// TIA Portal V17 export
// export: Created 2024-08-26T21:10:49.0093194Z, ExportSetting WithDefaults, DisplayName Totally Integrated Automation Portal, DisplayVersion V17 Update 7, DisplayName TIA Portal Openness, DisplayVersion V17 Update 7, DisplayName TIA Portal Version Control Interface, DisplayVersion V17, DisplayName SINAMICS Startdrive Advanced, DisplayVersion V17 SP2, DisplayName SINAMICS Startdrive G110M, G120, G120C, G120D, G120P, G115D, DisplayVersion V17 SP2, DisplayName SINAMICS Startdrive G130, G150, S120, S150, SINAMICS MV, S210, DisplayVersion V17 SP2, DisplayName STEP 7 Professional, DisplayVersion V17 Update 7, DisplayName STEP 7 Safety, DisplayVersion V17 Update 6, DisplayName WinCC Advanced / Unified PC, DisplayVersion V17 Update 7
FUNCTION "smartLightControl" : Void   // FC7, LAD
{ S7_Optimized_Access := 'TRUE' }
VERSION : 0.1
// stored: AutoNumber true, IsIECCheckEnabled false, SetENOAutomatically false, UDAEnableTagReadback false
   VAR_INPUT
      iRedSolid : Bool;
      iRedBlinking : Bool;
      iAmbarSolid : Bool;
      iAmbarBlinking : Bool;
      iGreenSolid : Bool;
      iGreenBlinking : Bool;
      iBlueSolid : Bool;
      iBlueBlinking : Bool;
   END_VAR
   VAR_OUTPUT
      byte0ColorAndBlink : Byte;   // Segment 1 and 2
      byte1ColorAndBlink : Byte;   // Segment 3
      byte2BuzzerType : Byte;
      byte3ModeSelect : Byte;
      byte4NumberOfSegments : Byte;
      byte5BlinkMode : Byte;
      byte6BlinkFreq : Byte;
      byte7BuzzerVolume : Byte;
   END_VAR
   VAR_TEMP
      segment1Color : Byte;
      segment2Color : Byte;
      segment3Color : Byte;
      colorsToDisplay : Word;
      numberOfColorsToDisplay : UInt;
      colorToAddToQueue : Word;
      positionsToMove : UInt;
   END_VAR
   VAR CONSTANT
      redColor : Byte := 2#0010;
      blueColor : Byte := 2#0100;
      ambarColor : Byte := 2#0101;
      greenColor : Byte := 2#0001;
      redBlinkingColor : Byte := 2#1010;
      blueBlinkingColor : Byte := 2#1100;
      ambarBlinkingColor : Byte := 2#1101;
      greenBlinkingColor : Byte := 2#1001;
   END_VAR
BEGIN

REGION Network 1: INIT
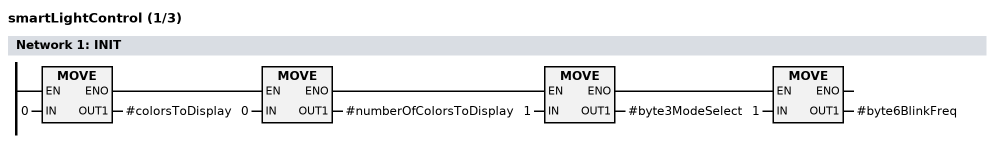
   RUNG wire#powerrail
      Move(in := 0, out1 => #colorsToDisplay)
      Move(in := 0, out1 => #numberOfColorsToDisplay)
      Move(in := 1, out1 => #byte3ModeSelect)
      Move(in := 1, out1 => #byte6BlinkFreq)
   END_RUNG
   // the same network as SCL:
   #colorsToDisplay := 0;
   #numberOfColorsToDisplay := 0;
   #byte3ModeSelect := 1;
   #byte6BlinkFreq := 1;
END_REGION

REGION Network 2: Select colors to display
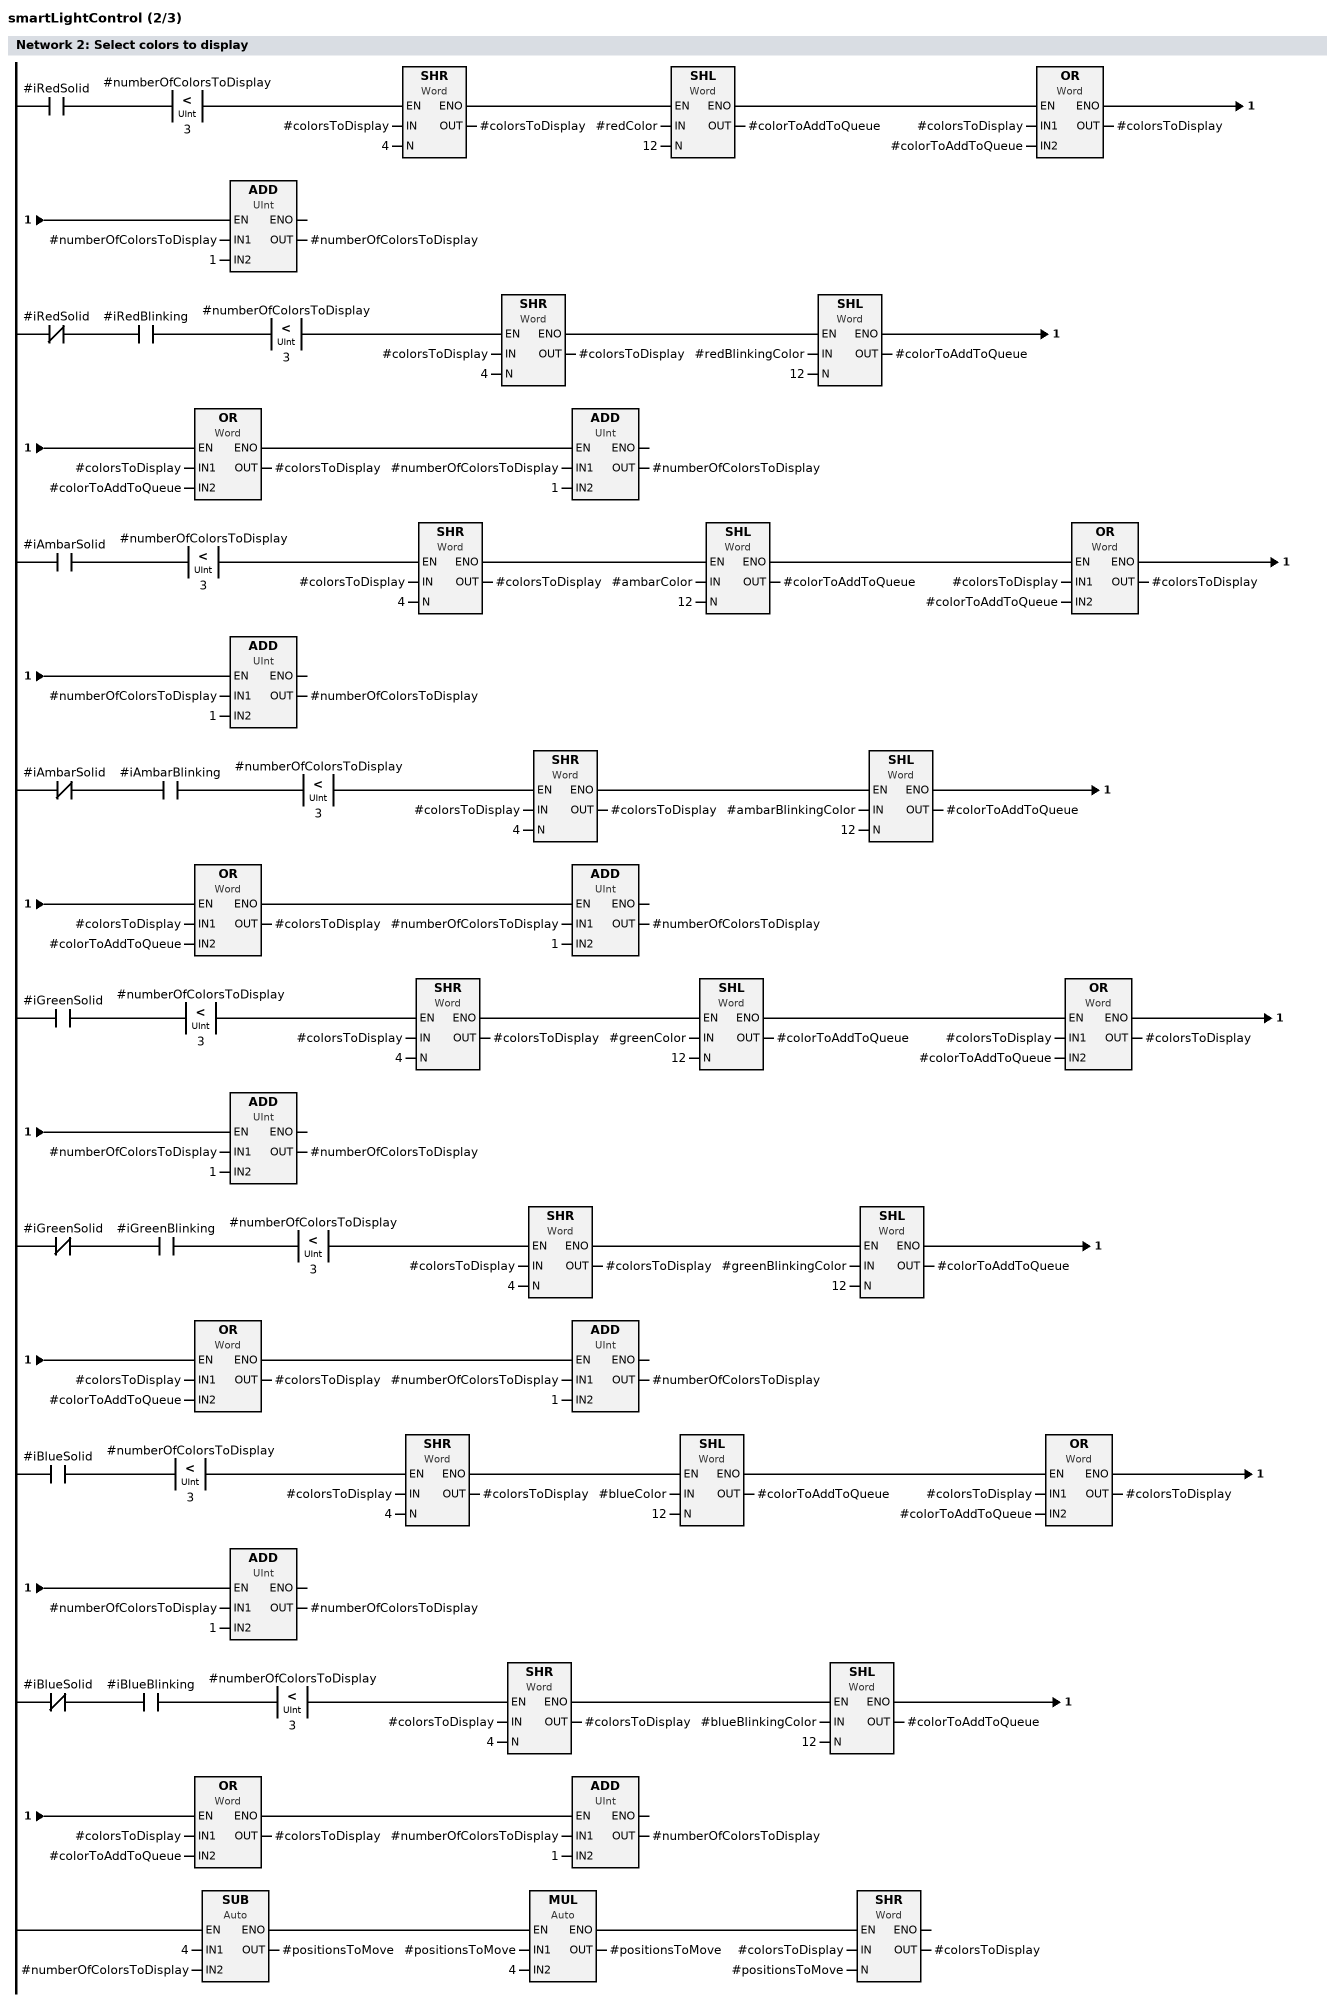
   IF #iRedSolid AND (#numberOfColorsToDisplay < 3) THEN
       #colorsToDisplay := SHR(IN := #colorsToDisplay, N := 4);
       #colorToAddToQueue := SHL(IN := #redColor, N := 12);
       #colorsToDisplay := #colorsToDisplay OR #colorToAddToQueue;
       #numberOfColorsToDisplay := #numberOfColorsToDisplay + 1;
   END_IF;
   IF NOT #iRedSolid AND #iRedBlinking AND (#numberOfColorsToDisplay < 3) THEN
       #colorsToDisplay := SHR(IN := #colorsToDisplay, N := 4);
       #colorToAddToQueue := SHL(IN := #redBlinkingColor, N := 12);
       #colorsToDisplay := #colorsToDisplay OR #colorToAddToQueue;
       #numberOfColorsToDisplay := #numberOfColorsToDisplay + 1;
   END_IF;
   IF #iAmbarSolid AND (#numberOfColorsToDisplay < 3) THEN
       #colorsToDisplay := SHR(IN := #colorsToDisplay, N := 4);
       #colorToAddToQueue := SHL(IN := #ambarColor, N := 12);
       #colorsToDisplay := #colorsToDisplay OR #colorToAddToQueue;
       #numberOfColorsToDisplay := #numberOfColorsToDisplay + 1;
   END_IF;
   IF NOT #iAmbarSolid AND #iAmbarBlinking AND (#numberOfColorsToDisplay < 3) THEN
       #colorsToDisplay := SHR(IN := #colorsToDisplay, N := 4);
       #colorToAddToQueue := SHL(IN := #ambarBlinkingColor, N := 12);
       #colorsToDisplay := #colorsToDisplay OR #colorToAddToQueue;
       #numberOfColorsToDisplay := #numberOfColorsToDisplay + 1;
   END_IF;
   IF #iGreenSolid AND (#numberOfColorsToDisplay < 3) THEN
       #colorsToDisplay := SHR(IN := #colorsToDisplay, N := 4);
       #colorToAddToQueue := SHL(IN := #greenColor, N := 12);
       #colorsToDisplay := #colorsToDisplay OR #colorToAddToQueue;
       #numberOfColorsToDisplay := #numberOfColorsToDisplay + 1;
   END_IF;
   IF NOT #iGreenSolid AND #iGreenBlinking AND (#numberOfColorsToDisplay < 3) THEN
       #colorsToDisplay := SHR(IN := #colorsToDisplay, N := 4);
       #colorToAddToQueue := SHL(IN := #greenBlinkingColor, N := 12);
       #colorsToDisplay := #colorsToDisplay OR #colorToAddToQueue;
       #numberOfColorsToDisplay := #numberOfColorsToDisplay + 1;
   END_IF;
   IF #iBlueSolid AND (#numberOfColorsToDisplay < 3) THEN
       #colorsToDisplay := SHR(IN := #colorsToDisplay, N := 4);
       #colorToAddToQueue := SHL(IN := #blueColor, N := 12);
       #colorsToDisplay := #colorsToDisplay OR #colorToAddToQueue;
       #numberOfColorsToDisplay := #numberOfColorsToDisplay + 1;
   END_IF;
   IF NOT #iBlueSolid AND #iBlueBlinking AND (#numberOfColorsToDisplay < 3) THEN
       #colorsToDisplay := SHR(IN := #colorsToDisplay, N := 4);
       #colorToAddToQueue := SHL(IN := #blueBlinkingColor, N := 12);
       #colorsToDisplay := #colorsToDisplay OR #colorToAddToQueue;
       #numberOfColorsToDisplay := #numberOfColorsToDisplay + 1;
   END_IF;
   #positionsToMove := 4 - #numberOfColorsToDisplay;
   #positionsToMove := #positionsToMove * 4;
   #colorsToDisplay := SHR(IN := #colorsToDisplay, N := #positionsToMove);
END_REGION

REGION Network 3: Send Colors to Byte 1 and 2
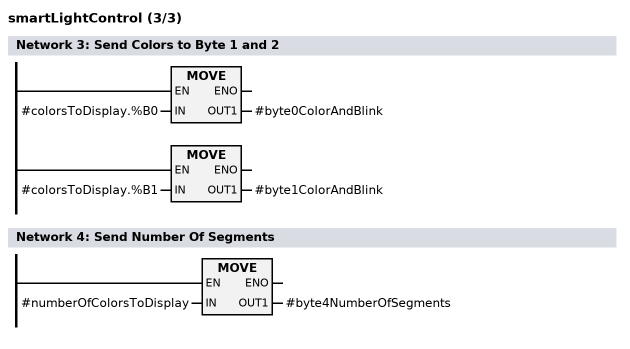
   RUNG wire#powerrail
      Move(in := #colorsToDisplay.%B0, out1 => #byte0ColorAndBlink)
   END_RUNG
   RUNG wire#powerrail
      Move(in := #colorsToDisplay.%B1, out1 => #byte1ColorAndBlink)
   END_RUNG
   // the same network as SCL:
   #byte0ColorAndBlink := #colorsToDisplay.%B0;
   #byte1ColorAndBlink := #colorsToDisplay.%B1;
END_REGION

REGION Network 4: Send Number Of Segments
   RUNG wire#powerrail
      Move(in := #numberOfColorsToDisplay, out1 => #byte4NumberOfSegments)
   END_RUNG
   // the same network as SCL:
   #byte4NumberOfSegments := #numberOfColorsToDisplay;
END_REGION
END_FUNCTION
